// TwinCAT 3 PLC project Untitled1
// ProgramVersion: 3.1.4024.0
// libraries:
//   Tc2_EtherCAT, * (Beckhoff Automation GmbH)
//   Tc2_MC2, * (Beckhoff Automation GmbH)
//   Tc2_MC2_Drive, * (Beckhoff Automation GmbH)
//   Tc2_NC, * (Beckhoff Automation GmbH)
//   Tc2_Standard, * (Beckhoff Automation GmbH)
//   Tc2_System, * (Beckhoff Automation GmbH)
//   Tc3_Module, * (Beckhoff Automation GmbH)
// project tree:
//   DUTs/ E_Manufacturer.TcDUT, ST_FeedbackOneType.TcDUT
//   FUNCTIONS/ FB_ToStringMotionState.TcPOU, FB_ToStringSelectedDrillingheadType.TcPOU
//   / GlobalTextList.TcGTLO, PlcTask.TcTTO, Visualization Manager.TcVMO (not stored), VISU_TASK.TcTTO
//   GVLs/ IO.TcGVL, Safety.TcGVL
//   POUs/ MAIN.TcPOU, Motion.TcPOU, TestFBSoERead.TcPOU, TestfbSoEWrite.TcPOU, TestFB_EcSetSlaveState.TcPOU, Toolchanger.TcPOU
//   VISUs/ Header.TcVIS, ImagePool.TcIPO (not stored), MainScreen.TcVIS, Motion.TcVIS, Nav.TcVIS, SelectDrillinghead.TcVIS
// real-time tasks:
//   TASK PlcTask: cycle T#10ms, priority 20, ADS port 350
//   TASK VISU_TASK: cycle T#200000us, priority 30, ADS port 351
// motion (NC):
//   TASK NC-Task 1 SAF: cycle T#2ms, priority 4, ADS port 501
//   TASK NC-Task 1 SVB: cycle T#10ms, priority 8, ADS port 511
//   AXIS Axis 1 (id 1)
//     General: UnitName=°
//     Dynamic: AccelerationMaximum=10000, DecelerationMaximum=10000, Acceleration=20000, Deceleration=20000, Jerk=134973
//     Velo: RefSearch=299.94, RefSync=299.94, SlowManual=1499.7, FastManual=8998.2, Fast=29994, Maximum=29994
//     PositionAreaControl: Enable=false
//     TargetPosControl: Enable=false
//     OtherSettings: AllowMotionCmdToSlave=true, AllowMotionCmdToExtSetGenAxis=true
//     encoder EncType=8
//       EncPara: ScaleFactorNumerator=360, ScaleFactorDenominator=1048576, MaxCount=#xffffffff
//     drive DrvType=9
//       DrvPara: MaxCount=#xffffffff, DriveControlDWord=#x00030100
//         Analog: VeloReferenz=32993.4, VeloScale=1.02400649589962, TorqueSetpointScale=10, ScaleFactorActTorque=0.1
//         TimeComp: TaskDelayCycles=1
//     controller CtrType=1
//       CtrPara: PriorControlFactor=1
//         PosDiffControl: Enable=false
//         Observer: BandWidth=20
// I/O:
//   DEVICE Device 2 (EtherCAT), AmsNetId 10.100.6.93.3.1
//     Term 9 (EK1100) [EK1100 EtherCAT Coupler (2A E-Bus)]
//       Term 10 (EL6900) [EL6900, TwinSAFE PLC]
//       Term 11 (EL1904) [EL1904, 4 Ch. Safety Input 24V, TwinSAFE]
//         modules: Module 1 (FSOES)
//       Term 12 (EL1104) [EL1104 4Ch. Dig. Input 24V, 3ms, Sensor Power]
//       Term 13 (EL2004) [EL2004 4Ch. Dig. Output 24V, 0.5A]
//       Term 15 (EL9011) [EL9011 End Terminal]
//     Drive 14 (AX5140-0000-0213) [AX5140-0000-0213 EtherCAT Drive (SoE, 1 Ch.)]
// variable links:
//   (this object) <-> Device 2 (EtherCAT)/Drive 14 (AX5140-0000-0213)
//     Drive/Inputs/In/nDataIn1 <-> AT/Following distance
//     Drive/Inputs/In/nDcOutputTime <-> InfoData/DcOutputShift
//     Drive/Inputs/In/nState1 <-> AT/Drive status word @bit 8
//     Drive/Inputs/In/nState2 <-> AT/Drive status word
//     Drive/Inputs/In/nState4 @bit 1 <-> WcState/InputToggle
//     Drive/Inputs/In/nState4 <-> WcState/WcState
//     Drive/Outputs/Out/nCtrl1 <-> MDT/Master control word @bit 8
//     Drive/Outputs/Out/nDataOut1 <-> MDT/Position command value
//     Enc/Inputs/In/nDataIn1 <-> AT/Position feedback 1 value
//     Enc/Inputs/In/nDcInputTime <-> InfoData/DcInputShift
//     Enc/Inputs/In/nState4 @bit 1 <-> WcState/InputToggle
//     Enc/Inputs/In/nState4 <-> WcState/WcState
//   Untitled1 Instance <-> Device 2 (EtherCAT)/Term 9 (EK1100)/Term 12 (EL1104)
//     PlcTask Inputs/Toolchanger.bToolChangerButton <-> Channel 1/Input
//   Untitled1 Instance <-> Device 2 (EtherCAT)/Term 9 (EK1100)/Term 13 (EL2004)
//     PlcTask Outputs/Toolchanger.bToolChangerCylinderIn <-> Channel 2/Output
//     PlcTask Outputs/Toolchanger.bToolChangerCylinderOut <-> Channel 1/Output
//   Untitled1 Instance <-> NC-Task 1 SAF/Axes/Axis 1
//     PlcTask Inputs/Motion.Axis1.NcToPlc <-> Outputs/ToPlc
//     PlcTask Outputs/Motion.Axis1.PlcToNc <-> Inputs/FromPlc

CONFIGURATION Untitled1
    RESOURCE PLC ON TwinCAT3
        TASK PlcTask(INTERVAL := T#10ms, PRIORITY := 20);
        TASK VISU_TASK(INTERVAL := T#200000us, PRIORITY := 30);
        PROGRAM MAIN WITH PlcTask : MAIN;
        PROGRAM VisuElems_Visu_Prg WITH VISU_TASK : VisuElems.Visu_Prg;
    END_RESOURCE
END_CONFIGURATION

// ---- DUTs/E_Manufacturer.TcDUT
{attribute 'qualified_only'}
{attribute 'strict'}
TYPE E_Manufacturer :
(
	Unknown_manufacturer := 0,
	Hengstler
);
END_TYPE

// ---- DUTs/ST_FeedbackOneType.TcDUT
TYPE ST_FeedbackOneType :
STRUCT
	Manufacturer : E_Manufacturer;



END_STRUCT
END_TYPE

// ---- GVLs/IO.TcGVL
{attribute 'qualified_only'}
VAR_GLOBAL
	
	bInAckSignal	AT %I* : BOOL;

END_VAR

// ---- GVLs/Safety.TcGVL
{attribute 'qualified_only'}
VAR_GLOBAL

	bSafetyErrorAck 	AT %Q* : BOOL;
	bAXSafetyErrorAck 	AT %Q* : BOOL;
	bSafetyRun			AT %Q* : BOOL;
	bSafetyRestart		AT %Q* : BOOL;

END_VAR

// ---- POUs/MAIN.TcPOU
PROGRAM MAIN
VAR
END_VAR

//Safety.bSafetyRestart 		:= IO.bInAckSignal;
//Safety.bSafetyErrorAck 		:= IO.bInAckSignal;
//Safety.bAXSafetyErrorAck 	:= IO.bInAckSignal;
//Safety.bSafetyRun 			:= TRUE;

Motion();
Toolchanger();
//TestfbSoEWrite();
//TestFBSoERead();
//TestFB_EcSetSlaveState();

END_PROGRAM

// ---- POUs/Motion.TcPOU
{attribute 'to_string'}
PROGRAM Motion
VAR
	// Digital inputs (Start/stop)
	iStartButton AT %I* : BOOL;
	iStopButton AT %I* 	: BOOL;
	
	bStartButton : BOOL;
	bStopButton : BOOL;
	
	bNone : BOOL;
	bV310 : BOOL;
	bV320 : BOOL;

	// Axis
	Axis1 : AXIS_REF;
	
	McPower : MC_Power;
	McReset : MC_Reset;
	McJogging : MC_Jog;
	McVelocity : MC_MoveVelocity;
	McStop : MC_Stop;
	MaxVelocity : LREAL;
	SetVelocity : LREAL;
	OverrideVelocity : LREAL;
	
	// States
	eMotionState : (Initial, StartDriveReset, WaitForDriveReset, DriveReady, StartMotor, StopMotor, Error);
	sMotionState : STRING;
	
	eSelectedDrillingheadType : (ToNone, None, ToV310, V310, ToV320, V320);
	sSelectedDrillingheadType : STRING;
	
END_VAR

//CurrentVelocityCmd := 1000.0;

MaxVelocity := 4000.0;
OverrideVelocity := SetVelocity/MaxVelocity * 100;

Axis1.ReadStatus();

//  Override := OverrideVelocity
McPower(Axis := Axis1, Enable := TRUE, Enable_Positive := TRUE, Enable_Negative := TRUE, Override := OverrideVelocity);
McReset(Axis := Axis1);
McJogging(Axis := Axis1);

// Motor state
FB_ToStringMotionState(_eMotionState := eMotionState,
						_sMotionState := sMotionState);

CASE eMotionState OF
	Initial:
		eMotionState := StartDriveReset;
		McReset(Axis := Axis1,Execute := FALSE);
	
	StartDriveReset:
		McReset(Axis := Axis1,Execute := TRUE);
		IF McReset.Done THEN
			eMotionState := WaitForDriveReset;
		ELSIF McReset.Error THEN
			eMotionState := Error;
		END_IF
	
	WaitForDriveReset:
		McReset(Axis := Axis1,Execute := FALSE);
		IF McPower.Status THEN
			eMotionState := DriveReady;
		END_IF
	
	DriveReady:
		IF bStartButton THEN
			eMotionState := StartMotor;
		END_IF
		
	StartMotor:
		McVelocity(Axis:=Axis1,
				Velocity:=MaxVelocity,
				Acceleration:=10000,
				Deceleration:=10000,
				Jerk:=100000,
				Direction:=MC_Direction.MC_Positive_Direction,
				Execute:=TRUE);
		
		IF bStopButton THEN
			McVelocity(Axis:=Axis1, Execute:=FALSE);
			eMotionState := StopMotor;
		END_IF
		
	StopMotor:
		McStop(Axis:=Axis1, Execute:=TRUE);
		
		IF bStartButton THEN
			McStop(Axis:=Axis1, Execute:=FALSE);
			eMotionState := StartMotor;
		END_IF
		
	Error:
		McReset(Axis := Axis1,Execute := FALSE);
		eMotionState := Initial;
	
END_CASE


// Drilling head selection
FB_ToStringSelectedDrillingheadType(_eSelectedDrillingheadType := eSelectedDrillingheadType,
									_sSelectedDrillingheadType := sSelectedDrillingheadType);

IF Axis1.Status.HasBeenStopped THEN
	IF bNone THEN
		eSelectedDrillingheadType := ToNone;
	
	ELSIF bV310 THEN
		eSelectedDrillingheadType := ToV310;
		
	ELSIF bV320 THEN
		eSelectedDrillingheadType := ToV320;
	
	END_IF
END_IF

									
									
									
									

									
									
CASE eSelectedDrillingHeadType OF
	ToNone:
	
	
	None:
	
	
	ToV310:
	
	
	V310:
	
	
	ToV320:
	
	
	V320:
	
	
END_CASE

END_PROGRAM

// ---- FUNCTIONS/FB_ToStringMotionState.TcPOU
FUNCTION FB_ToStringMotionState
VAR_INPUT
	_eMotionState : INT;
	_sMotionState : REFERENCE TO STRING;
END_VAR
VAR
END_VAR

IF _eMotionState = 0 THEN
	_sMotionState := 'Initial';
	
ELSIF _eMotionState = 1 THEN
	_sMotionState := 'StartDriveReset';
	
ELSIF _eMotionState = 2 THEN
	_sMotionState := 'WaitForDriveReset';
	
ELSIF _eMotionState = 3 THEN
	_sMotionState := 'DriveReady';
	
ELSIF _eMotionState = 4 THEN
	_sMotionState := 'StartMotor';
	
ELSIF _eMotionState = 5 THEN
	_sMotionState := 'StopMotor';

ELSIF _eMotionState = 6 THEN
	_sMotionState := 'Error';		

END_IF

END_FUNCTION

// ---- FUNCTIONS/FB_ToStringSelectedDrillingheadType.TcPOU
FUNCTION FB_ToStringSelectedDrillingheadType
VAR_INPUT
	_eSelectedDrillingheadType : INT;
	_sSelectedDrillingheadType : REFERENCE TO STRING;
END_VAR
VAR
END_VAR

IF _eSelectedDrillingheadType = 0 THEN
	_sSelectedDrillingheadType := 'ToNone';
	
ELSIF _eSelectedDrillingheadType = 1 THEN
	_sSelectedDrillingheadType := 'None';
	
ELSIF _eSelectedDrillingheadType = 2 THEN
	_sSelectedDrillingheadType := 'ToV310';
	
ELSIF _eSelectedDrillingheadType = 3 THEN
	_sSelectedDrillingheadType := 'V310';
	
ELSIF _eSelectedDrillingheadType = 4 THEN
	_sSelectedDrillingheadType := 'ToV320';
	
ELSIF _eSelectedDrillingheadType = 5 THEN
	_sSelectedDrillingheadType := 'V320';	

END_IF

END_FUNCTION

// ---- POUs/Toolchanger.TcPOU
PROGRAM Toolchanger
VAR
	bToolChangerButton 			AT %I*		: BOOL;		// Green push-button on the frame
	
	bToolChangerCylinderOut 	AT %Q*	: BOOL;		// 5/3 Monovalve OUT
	bToolChangerCylinderIn		AT %Q*	: BOOL;		// 5/3 Monovalve IN
END_VAR

IF bToolChangerButton AND Motion.Axis1.Status.HasBeenStopped THEN
	bToolChangerCylinderOut := FALSE;
	bToolChangerCylinderIn := TRUE;
	
ELSE
	bToolChangerCylinderOut := TRUE;
	bToolChangerCylinderIn := FALSE;
	
END_IF

END_PROGRAM

// ---- POUs/TestFBSoERead.TcPOU
PROGRAM TestFBSoERead
VAR
	fbSoERead : FB_SoERead;
	nTorqueLimit : UINT;
	
	bExecute : BOOL;
	stFeedbackOneType : ST_FeedbackOneType;
END_VAR





fbSoERead(
		Axis:= Motion.Axis1, 
		NetId:= '10.100.6.93.1.1', 
		Idn:= P_0_IDNs+150, 
		Element:= 16#40, 
		pDstBuf:= ADR(stFeedbackOneType), 
		BufLen:= SIZEOF(stFeedbackOneType), 
		Execute:= bExecute, 
		Timeout:= , 
		Busy=> , 
		Error=> , 
		AdsErrId=> , 
		SercosErrId=> , 
		Attribute=> );

END_PROGRAM

// ---- POUs/TestfbSoEWrite.TcPOU
PROGRAM TestfbSoEWrite
VAR
	fbSoEWrite : FB_SoEWrite;
	nTorqueLimit : UINT := 980;
	
	bExecute : BOOL;
	stFeedbackOneType : ST_FeedbackOneType;
END_VAR


stFeedbackOneType.Manufacturer := E_Manufacturer.Hengstler;

fbSoEWrite(
	Axis:= Motion.Axis1, 
	NetId:= '10.100.6.93.1.1', 
	Idn:= S_0_IDNs+150, 
	Element:= 16#40, 
	pSrcBuf:= ADR(stFeedbackOneType), 
	BufLen:= SIZEOF(stFeedbackOneType), 
	Execute:= bExecute, 
	Timeout:= , 
	Password:= , 
	Busy=> , 
	Error=> , 
	AdsErrId=> , 
	SercosErrId=> );

END_PROGRAM

// ---- POUs/TestFB_EcSetSlaveState.TcPOU
PROGRAM TestFB_EcSetSlaveState
VAR
	fbEcSetSlaveState 	: FB_EcSetSlaveState;
	sNetId          	: T_AmsNetId:= '10.100.6.93.3.1';
	nSlaveAddr      	: UINT := 1006;
	bExecute        	: BOOL;
	tTimeout   			: TIME := T#10S;
	reqState   			: WORD;
END_VAR

fbEcSetSlaveState(
				sNetId:= sNetId, 
				nSlaveAddr:= nSlaveAddr, 
				bExecute:= bExecute, 
				tTimeout:= tTimeout, 
				reqState:= reqState, 
				bBusy=> , 
				bError=> , 
				nErrId=> , 
				currState=> );

END_PROGRAM

// ---- GlobalTextList.TcGTLO
TEXTLIST GlobalTextList
  912 = '%5.2f'
  525 = '%s'
  734 = 'Actual motion state'
  322 = 'Actual Velocity'
  717 = 'bStartButton'
  130 = 'bStopButton'
  906 = 'MAIN'
  608 = 'MAIN SCREEN'
  875 = 'Motion'
  243 = 'None'
  590 = 'Select Drillinghead'
  443 = 'Selected Drillinghead'
  804 = 'Set Velocity'
  582 = 'TO MOTION'
  194 = 'TO SELECT DRILLINGHEAD'
  907 = 'V310'
  182 = 'V320'
END_TEXTLIST

// ---- VISUs/Header.TcVIS
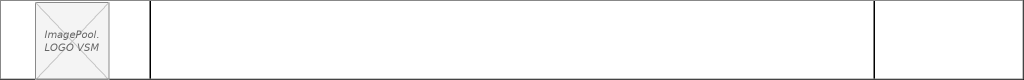
VISUALIZATION Header  // 1024x80
    Rectangle (0,0 150x80)
    Rectangle (150,0 724x80)
    Rectangle (874,0 150x80)
    Image (35,2 74x78), image: ImagePool.LOGO VSM
END_VISUALIZATION

// ---- VISUs/MainScreen.TcVIS
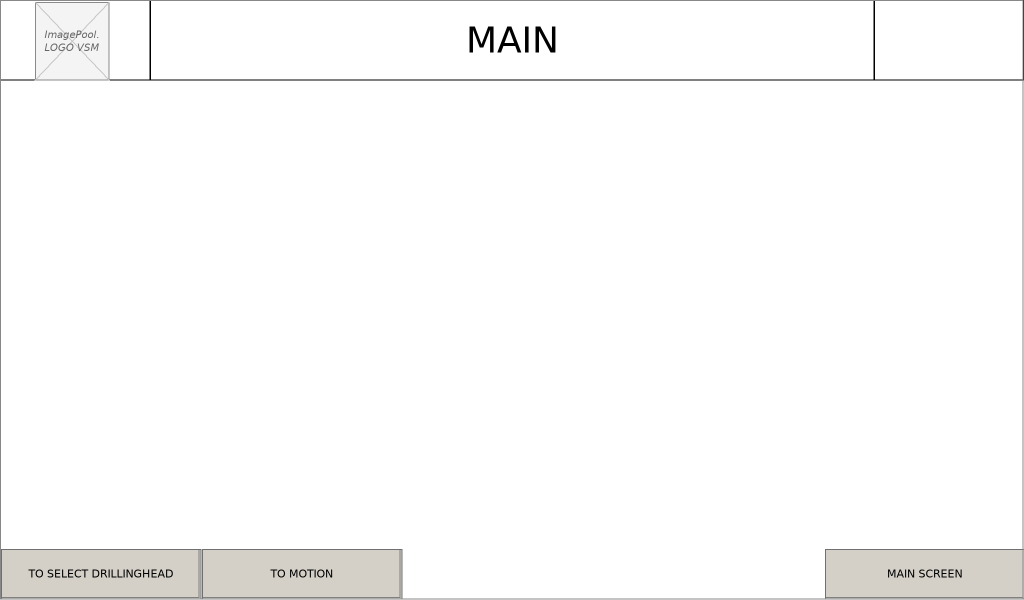
VISUALIZATION MainScreen  // 1024x600
    Frame (0,0 1024x80)
        shows Header()
    Frame (1,549 1024x50)
        shows Nav()
    Label (334,16 357x48), "MAIN"
END_VISUALIZATION

// ---- VISUs/Motion.TcVIS
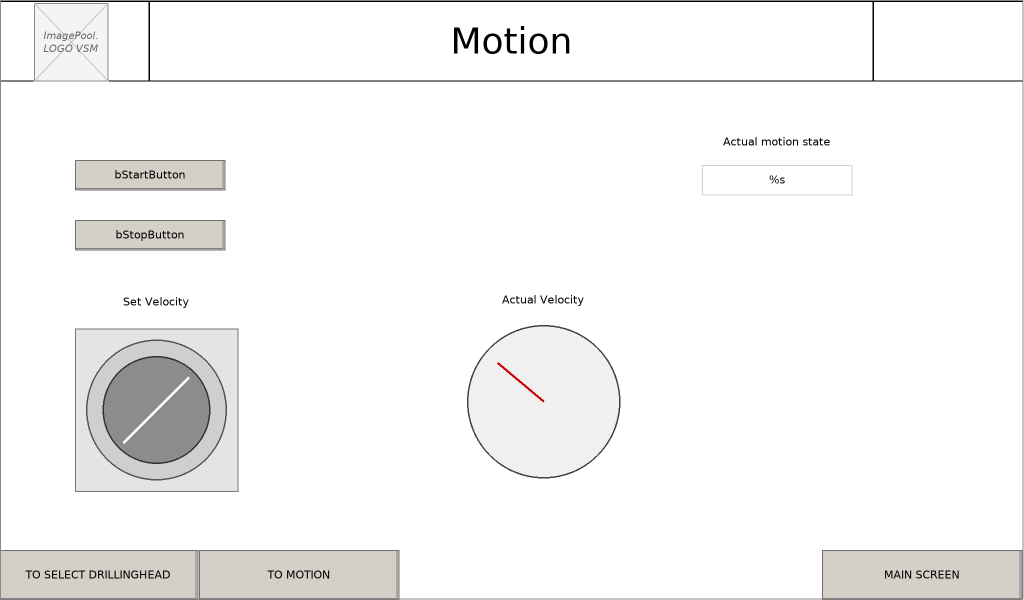
VISUALIZATION Motion  // 1024x600
    Frame (-1,1 1024x80)
        shows Header()
    Frame (-2,550 1024x50)
        shows Nav()
    Label (333,17 357x48), "Motion"
    Textfield (702,165 150x30), "%s", text variable: Motion.sMotionState
    Label (702,127 150x30), "Actual motion state"
    Button (75,160 150x30), "bStartButton"
        OnMouseDown: execute { Motion.bStartButton := TRUE; }
        OnMouseUp: execute { Motion.bStartButton := FALSE; }
    Button (75,220 150x30), "bStopButton"
        OnMouseDown: execute { Motion.bStopButton := TRUE; }
        OnMouseUp: execute { Motion.bStopButton := FALSE; }
    Potentiometer360 (75,325 163x170), variable: Motion.SetVelocity, style: Potentiometer-Potentiometer360-Gray, scale format: %.1f, scale 0..4000
        p2431819421: Outside
    Meter360 (465,325 157x153), value: Motion.Axis1.NcToPlc.ActVelo, style: Meter-Meter360-Gray, scale format: %5.2f, scale 0..4000
    Label (81,287 150x30), "Set Velocity"
    Label (468,285 150x30), "Actual Velocity"
END_VISUALIZATION

// ---- VISUs/Nav.TcVIS
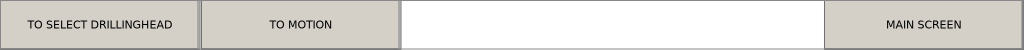
VISUALIZATION Nav  // 1024x50
    Button (0,0 200x50), "TO SELECT DRILLINGHEAD"
        OnMouseDown: change screen: SelectDrillinghead
    Button (201,0 200x50), "TO MOTION"
        OnMouseDown: change screen: Motion
    Button (824,0 200x50), "MAIN SCREEN"
        OnMouseDown: change screen: MainScreen
END_VISUALIZATION

// ---- VISUs/SelectDrillinghead.TcVIS
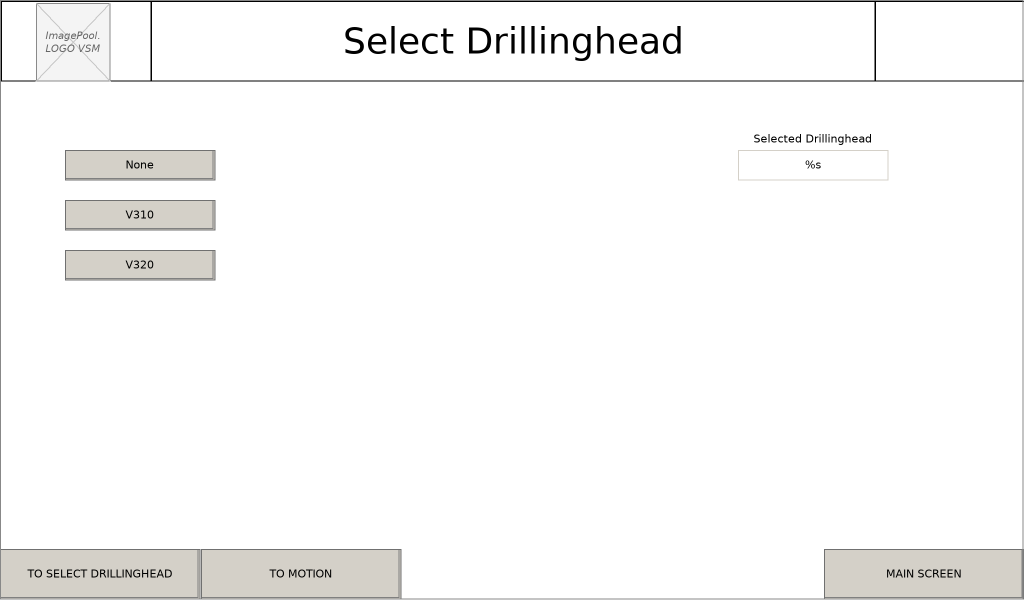
VISUALIZATION SelectDrillinghead  // 1024x600
    Frame (1,1 1024x80)
        shows Header()
    Frame (0,549 1024x50)
        shows Nav()
    Label (335,17 357x48), "Select Drillinghead"
    Textfield (738,150 150x30), "%s", text variable: Motion.sSelectedDrillingheadType
    Label (738,124 150x30), "Selected Drillinghead"
    Button (65,150 150x30), "None"
        OnMouseDown: execute { Motion.bNone := TRUE; }
        OnMouseUp: execute { Motion.bNone := FALSE; }
    Button (65,200 150x30), "V310"
        OnMouseDown: execute { Motion.bV310 := TRUE; }
        OnMouseUp: execute { Motion.bV310 := FALSE; }
    Button (65,250 150x30), "V320"
        OnMouseDown: execute { Motion.bV320 := TRUE; }
        OnMouseUp: execute { Motion.bV320 := FALSE; }
END_VISUALIZATION
